// TIA Portal V15.1 export
// export: Created 2024-06-21T08:41:07.4189134Z, ExportSetting WithDefaults, DisplayName Totally Integrated Automation Portal, DisplayVersion V15.1 Update 5, DisplayName TIA Portal Openness, DisplayVersion V15.1 Update 5, DisplayName SINAMICS Startdrive Advanced, DisplayVersion V15.1, DisplayName G130, G150, S120, S150, SINAMICS MV, S210, DisplayVersion V15.1, DisplayName G110M, G120, G120C, G120D, G120P, DisplayVersion V15.1, DisplayName STEP 7 Professional, DisplayVersion V15.1 Update 5, DisplayName STEP 7 Safety, DisplayVersion V15.1, DisplayName WinCC Professional, DisplayVersion V15.1 Update 5, DisplayName SIMATIC Visualization Architect, DisplayVersion V15.1
FUNCTION_BLOCK "LGBKP400"   // FB6660, FBD
TITLE = KP400 handling
{ S7_Optimized_Access := 'FALSE' }
AUTHOR : VCG
FAMILY : OPanel
VERSION : 1.0
// ================================================================================
// This module handles the modezone OP.
// Interlocking between OP's in the same modezone
// User interaction between the modezone and the interface
// ================================================================================
// 2021-07-26
// stored: AutoNumber false, IsIECCheckEnabled false, SetENOAutomatically False, UDAEnableTagReadback false
   VAR_INPUT
      I_OP_ID { ExternalAccessible := 'False'; ExternalVisible := 'False'; ExternalWritable := 'False'} : Int;   // Unique OP identification in the group
      I_ActiveHMI { ExternalAccessible := 'False'; ExternalVisible := 'False'; ExternalWritable := 'False'} : Int;   // Active HMI in the Modeselector
      I_ExtPBSet { ExternalAccessible := 'False'; ExternalVisible := 'False'; ExternalWritable := 'False'} : Bool;   // External PB set
      I_ExtPBReset { ExternalAccessible := 'False'; ExternalVisible := 'False'; ExternalWritable := 'False'} : Bool;   // External PB reset
   END_VAR
   VAR_OUTPUT
      O_ASSelected { ExternalAccessible := 'False'; ExternalVisible := 'False'; ExternalWritable := 'False'} : Bool;
      O_LampTest { ExternalAccessible := 'False'; ExternalVisible := 'False'; ExternalWritable := 'False'} : Bool;
      O_AutoModeSel { ExternalAccessible := 'False'; ExternalVisible := 'False'; ExternalWritable := 'False'} : Bool;
      O_ManualModeSel { ExternalAccessible := 'False'; ExternalVisible := 'False'; ExternalWritable := 'False'} : Bool;
      O_ResetSeq { ExternalAccessible := 'False'; ExternalVisible := 'False'; ExternalWritable := 'False'} : Bool;
      O_Start { ExternalAccessible := 'False'; ExternalVisible := 'False'; ExternalWritable := 'False'} : Bool;
      O_AlarmReset { ExternalAccessible := 'False'; ExternalVisible := 'False'; ExternalWritable := 'False'} : Bool;
      O_HighSpeed { ExternalAccessible := 'False'; ExternalVisible := 'False'; ExternalWritable := 'False'} : Bool;
      O_MovCode { ExternalAccessible := 'False'; ExternalVisible := 'False'; ExternalWritable := 'False'} : Int;
   END_VAR
   VAR_IN_OUT
      IO_GroupInterlock { ExternalAccessible := 'False'; ExternalVisible := 'False'; ExternalWritable := 'False'} : Int;   // Is this OP selected? Refers to the interlocking word of this group
      H_HMI : "H_HMI";
      H_GBKP400 : "H_GBKP400";
      IO_Modes : "Modes";   // Modes IO
   END_VAR
   VAR DB_SPECIFIC
      OP_Selected { ExternalAccessible := 'False'; ExternalVisible := 'False'; ExternalWritable := 'False'} : Bool;
      OP_Selected_NE { ExternalAccessible := 'False'; ExternalVisible := 'False'; ExternalWritable := 'False'} : Bool;
      FK_F1_Pressed { ExternalAccessible := 'False'; ExternalVisible := 'False'; ExternalWritable := 'False'} : Bool;
      FK_F2_Pressed { ExternalAccessible := 'False'; ExternalVisible := 'False'; ExternalWritable := 'False'} : Bool;
      FK_F3_Pressed { ExternalAccessible := 'False'; ExternalVisible := 'False'; ExternalWritable := 'False'} : Bool;
      FK_F4_Pressed { ExternalAccessible := 'False'; ExternalVisible := 'False'; ExternalWritable := 'False'} : Bool;
      FK_F5_Pressed { ExternalAccessible := 'False'; ExternalVisible := 'False'; ExternalWritable := 'False'} : Bool;   // Main Pressed
      FK_F6_Pressed { ExternalAccessible := 'False'; ExternalVisible := 'False'; ExternalWritable := 'False'} : Bool;   // Auto Pressed
      FK_F7_Pressed { ExternalAccessible := 'False'; ExternalVisible := 'False'; ExternalWritable := 'False'} : Bool;   // Man Pressed
      FK_F8_Pressed { ExternalAccessible := 'False'; ExternalVisible := 'False'; ExternalWritable := 'False'} : Bool;   // Step Pressed
      FK_F1_Pressed_hPE { ExternalAccessible := 'False'; ExternalVisible := 'False'; ExternalWritable := 'False'} : Bool;
      FK_F2_Pressed_hPE { ExternalAccessible := 'False'; ExternalVisible := 'False'; ExternalWritable := 'False'} : Bool;
      FK_F3_Pressed_hPE { ExternalAccessible := 'False'; ExternalVisible := 'False'; ExternalWritable := 'False'} : Bool;
      FK_F4_Pressed_hPE { ExternalAccessible := 'False'; ExternalVisible := 'False'; ExternalWritable := 'False'} : Bool;
      FK_F5_Pressed_hPE { ExternalAccessible := 'False'; ExternalVisible := 'False'; ExternalWritable := 'False'} : Bool;
      FK_F6_Pressed_hPE { ExternalAccessible := 'False'; ExternalVisible := 'False'; ExternalWritable := 'False'} : Bool;
      FK_F7_Pressed_hPE { ExternalAccessible := 'False'; ExternalVisible := 'False'; ExternalWritable := 'False'} : Bool;
      FK_F8_Pressed_hPE { ExternalAccessible := 'False'; ExternalVisible := 'False'; ExternalWritable := 'False'} : Bool;
      FK_F1_Pressed_PE { ExternalAccessible := 'False'; ExternalVisible := 'False'; ExternalWritable := 'False'} : Bool;
      FK_F2_Pressed_PE { ExternalAccessible := 'False'; ExternalVisible := 'False'; ExternalWritable := 'False'} : Bool;
      FK_F3_Pressed_PE { ExternalAccessible := 'False'; ExternalVisible := 'False'; ExternalWritable := 'False'} : Bool;
      FK_F4_Pressed_PE { ExternalAccessible := 'False'; ExternalVisible := 'False'; ExternalWritable := 'False'} : Bool;
      FK_F5_Pressed_PE { ExternalAccessible := 'False'; ExternalVisible := 'False'; ExternalWritable := 'False'} : Bool;
      FK_F6_Pressed_PE { ExternalAccessible := 'False'; ExternalVisible := 'False'; ExternalWritable := 'False'} : Bool;
      FK_F7_Pressed_PE { ExternalAccessible := 'False'; ExternalVisible := 'False'; ExternalWritable := 'False'} : Bool;
      FK_F8_Pressed_PE { ExternalAccessible := 'False'; ExternalVisible := 'False'; ExternalWritable := 'False'} : Bool;
      MainScreenActive { ExternalAccessible := 'False'; ExternalVisible := 'False'; ExternalWritable := 'False'} : Bool;
      AutoScreenActive { ExternalAccessible := 'False'; ExternalVisible := 'False'; ExternalWritable := 'False'} : Bool;
      AutoSelScreenActive { ExternalAccessible := 'False'; ExternalVisible := 'False'; ExternalWritable := 'False'} : Bool;
      ManScreenActive { ExternalAccessible := 'False'; ExternalVisible := 'False'; ExternalWritable := 'False'} : Bool;
      MVTScreenActive { ExternalAccessible := 'False'; ExternalVisible := 'False'; ExternalWritable := 'False'} : Bool;
      ProdScreenActive { ExternalAccessible := 'False'; ExternalVisible := 'False'; ExternalWritable := 'False'} : Bool;
      SSScreenActive { ExternalAccessible := 'False'; ExternalVisible := 'False'; ExternalWritable := 'False'} : Bool;
      SSSelScreenActive { ExternalAccessible := 'False'; ExternalVisible := 'False'; ExternalWritable := 'False'} : Bool;
      Request_Logout { ExternalAccessible := 'False'; ExternalVisible := 'False'; ExternalWritable := 'False'} : Bool;
      OP_TimeoutInput { ExternalAccessible := 'False'; ExternalVisible := 'False'; ExternalWritable := 'False'} : Bool;
      AutoSel { ExternalAccessible := 'False'; ExternalVisible := 'False'; ExternalWritable := 'False'} : Bool;
      ManualSel { ExternalAccessible := 'False'; ExternalVisible := 'False'; ExternalWritable := 'False'} : Bool;
      AutoSel_PE { ExternalAccessible := 'False'; ExternalVisible := 'False'; ExternalWritable := 'False'} : Bool;
      ManSel_PE { ExternalAccessible := 'False'; ExternalVisible := 'False'; ExternalWritable := 'False'} : Bool;
      AlarmReset { ExternalAccessible := 'False'; ExternalVisible := 'False'; ExternalWritable := 'False'} : Bool;
      Start { ExternalAccessible := 'False'; ExternalVisible := 'False'; ExternalWritable := 'False'} : Bool;
      ResetTM { ExternalAccessible := 'False'; ExternalVisible := 'False'; ExternalWritable := 'False'} : Bool;
      ResetSeq { ExternalAccessible := 'False'; ExternalVisible := 'False'; ExternalWritable := 'False'} : Bool;
      AutoMode { ExternalAccessible := 'False'; ExternalVisible := 'False'; ExternalWritable := 'False'} : Bool;
      StepMode { ExternalAccessible := 'False'; ExternalVisible := 'False'; ExternalWritable := 'False'} : Bool;
      ManualMode { ExternalAccessible := 'False'; ExternalVisible := 'False'; ExternalWritable := 'False'} : Bool;
      Alarm { ExternalAccessible := 'False'; ExternalVisible := 'False'; ExternalWritable := 'False'} : Bool;
      STAT4 { ExternalAccessible := 'False'; ExternalVisible := 'False'; ExternalWritable := 'False'} : Bool;
      STAT5 { ExternalAccessible := 'False'; ExternalVisible := 'False'; ExternalWritable := 'False'} : Bool;
      STAT6 { ExternalAccessible := 'False'; ExternalVisible := 'False'; ExternalWritable := 'False'} : Bool;
      STAT7 { ExternalAccessible := 'False'; ExternalVisible := 'False'; ExternalWritable := 'False'} : Bool;
      STAT8 { ExternalAccessible := 'False'; ExternalVisible := 'False'; ExternalWritable := 'False'} : Bool;
      STAT9 { ExternalAccessible := 'False'; ExternalVisible := 'False'; ExternalWritable := 'False'} : Bool;
      STAT10 { ExternalAccessible := 'False'; ExternalVisible := 'False'; ExternalWritable := 'False'} : Bool;
      STAT11 { ExternalAccessible := 'False'; ExternalVisible := 'False'; ExternalWritable := 'False'} : Bool;
      STAT12 { ExternalAccessible := 'False'; ExternalVisible := 'False'; ExternalWritable := 'False'} : Bool;
      OP_ScreenWanted { ExternalAccessible := 'False'; ExternalVisible := 'False'; ExternalWritable := 'False'} : Int;
      MovCode { ExternalAccessible := 'False'; ExternalVisible := 'False'; ExternalWritable := 'False'} : Int;
      MovCodeCalculation { ExternalAccessible := 'False'; ExternalVisible := 'False'; ExternalWritable := 'False'} : Int;
      ProdStatus { ExternalAccessible := 'False'; ExternalVisible := 'False'; ExternalWritable := 'False'} : Int;   // Production Mode
      ActiveMode { ExternalAccessible := 'False'; ExternalVisible := 'False'; ExternalWritable := 'False'} : Int;
      OPMode { ExternalAccessible := 'False'; ExternalVisible := 'False'; ExternalWritable := 'False'} : Int;
      GroupInterlock { ExternalAccessible := 'False'; ExternalVisible := 'False'; ExternalWritable := 'False'} : Int;
      ResetOP { ExternalAccessible := 'False'; ExternalVisible := 'False'; ExternalWritable := 'False'} : Bool;
      Edge { ExternalAccessible := 'False'; ExternalVisible := 'False'; ExternalWritable := 'False'} : Array[1..10] of Bool;
   END_VAR
   VAR
      Timer_Timeout_Input { ExternalAccessible := 'False'; ExternalVisible := 'False'; ExternalWritable := 'False'} : "LTimer";
   END_VAR
   VAR DB_SPECIFIC
      ModeEdge { ExternalAccessible := 'False'; ExternalVisible := 'False'; ExternalWritable := 'False'} : Array[1..10] of Bool;
   END_VAR
   VAR_TEMP
      OP_CommsDB : Int;
   END_VAR
   // // H_GBKP400.OPStatus : KP400 status
   // // H_GBKP400.OPMode : KP400 mode
   // // H_GBKP400.OPAdditional : KP400 additional info
   VAR_TEMP   // added for the SCL form of the ladder/FBD networks
      _w1 : Bool;
   END_VAR
BEGIN

REGION Network 1: **** 1 - Inputs **** Is this KP400 active?
   // Is this KP400 active?
   // IF yes:
   //  * Set OP as active 
   // IF not:
   //  * Reset flowcode
   //  * Reset MVT code
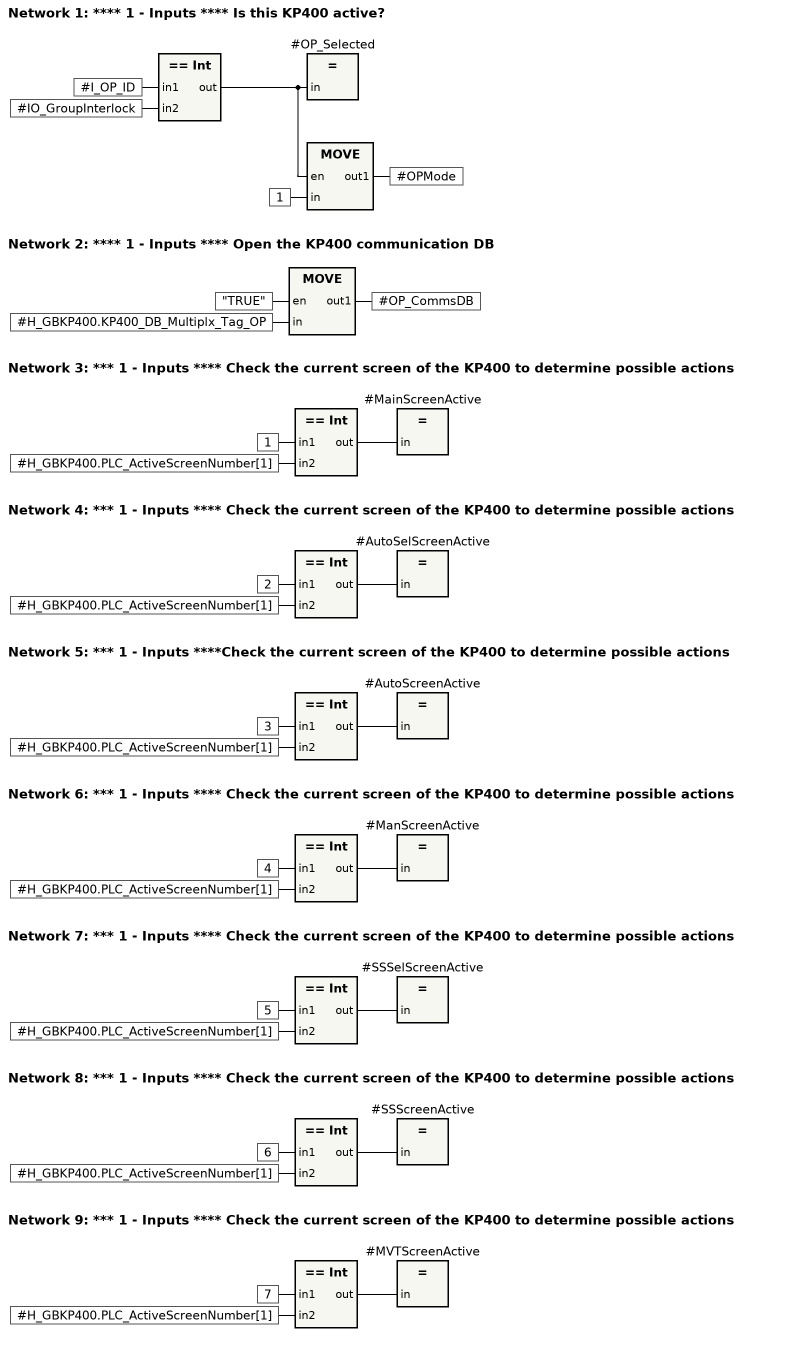
   #OP_Selected := #I_OP_ID = #IO_GroupInterlock;
   IF #OP_Selected THEN #OPMode := 1; END_IF;
END_REGION

REGION Network 2: **** 1 - Inputs **** Open the KP400 communication DB
   // Open the KP400 communication DB
   IF "TRUE" THEN #OP_CommsDB := #H_GBKP400.KP400_DB_Multiplx_Tag_OP; END_IF;
END_REGION

REGION Network 3: *** 1 - Inputs **** Check the current screen of the KP400 to determine possible actions
   // Check the current screen of the KP400 to determine possible actions
   //  1: Menu_Main
   //  2: Menu_Auto_Sel
   //  3: Menu_Auto
   //  4: Menu_Man
   //  5: Menu_SS_Sel
   //  6: Menu_SS
   //  7: Menu_MVT
   //  8: Menu_Flow
   //  9: Menu_Prod
   #MainScreenActive := 1 = #H_GBKP400.PLC_ActiveScreenNumber[1];
END_REGION

REGION Network 4: *** 1 - Inputs **** Check the current screen of the KP400 to determine possible actions
   // Check the current screen of the KP400 to determine possible actions
   //  2: Menu_Auto_Sel
   #AutoSelScreenActive := 2 = #H_GBKP400.PLC_ActiveScreenNumber[1];
END_REGION

REGION Network 5: *** 1 - Inputs ****Check the current screen of the KP400 to determine possible actions
   // Check the current screen of the KP400  to determine possible actions
   //  3: Menu_Auto
   #AutoScreenActive := 3 = #H_GBKP400.PLC_ActiveScreenNumber[1];
END_REGION

REGION Network 6: *** 1 - Inputs **** Check the current screen of the KP400 to determine possible actions
   // Check the current screen of the KP400  to determine possible actions
   //  4: Menu_Man
   #ManScreenActive := 4 = #H_GBKP400.PLC_ActiveScreenNumber[1];
END_REGION

REGION Network 7: *** 1 - Inputs **** Check the current screen of the KP400 to determine possible actions
   // Check the current screen of the KP400  to determine possible actions
   //  5: Menu_SS_Sel
   #SSSelScreenActive := 5 = #H_GBKP400.PLC_ActiveScreenNumber[1];
END_REGION

REGION Network 8: *** 1 - Inputs **** Check the current screen of the KP400 to determine possible actions
   // Check the current screen of the KP400  to determine possible actions
   //  6: Menu_SS
   #SSScreenActive := 6 = #H_GBKP400.PLC_ActiveScreenNumber[1];
END_REGION

REGION Network 9: *** 1 - Inputs **** Check the current screen of the KP400 to determine possible actions
   // Check the current screen of the KP400  to determine possible actions
   //  7: Menu_MVT
   #MVTScreenActive := 7 = #H_GBKP400.PLC_ActiveScreenNumber[1];
END_REGION

REGION Network 10: *** 1 - Inputs **** Check the current screen of the KP400 to determine possible actions
   // Check the current screen of the KP400  to determine possible actions
   //  9: Menu_Prod
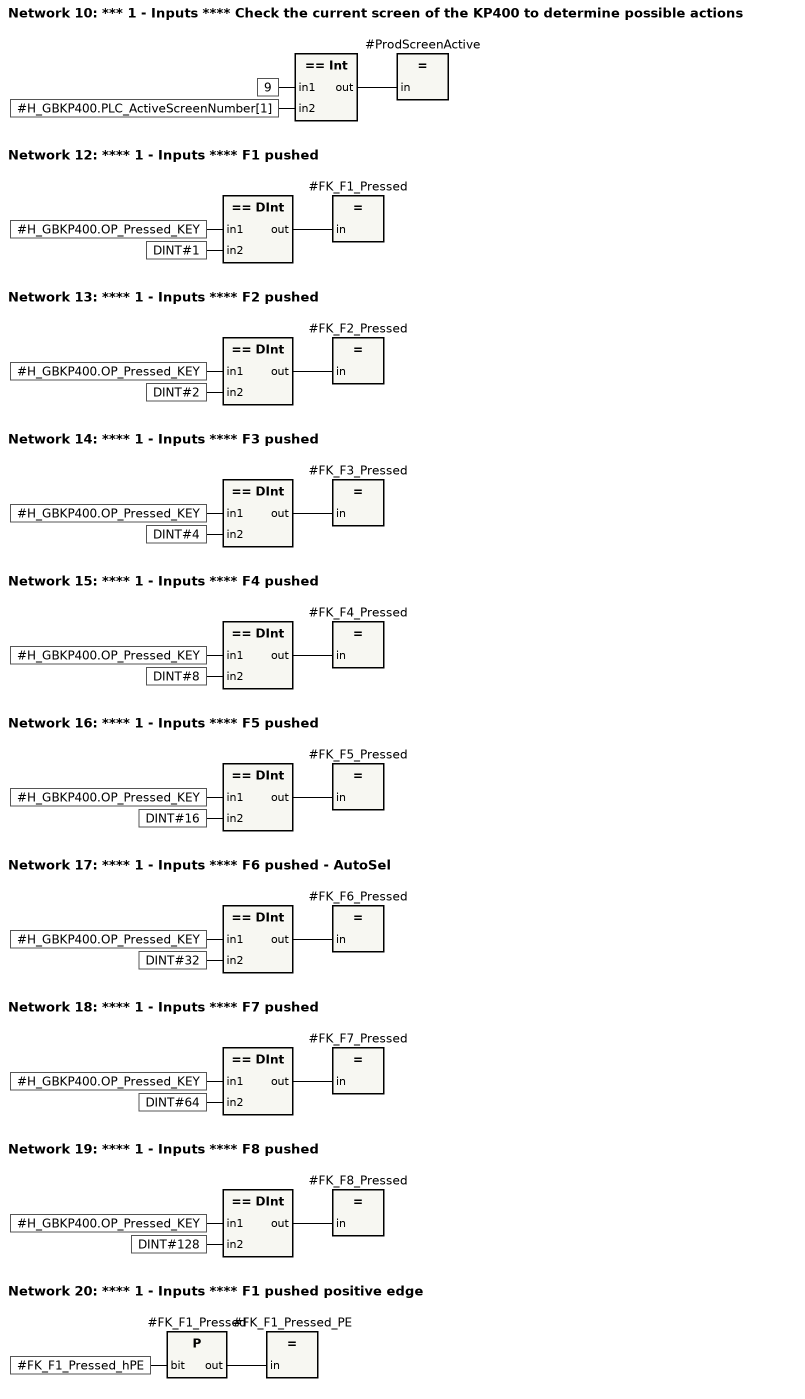
   #ProdScreenActive := 9 = #H_GBKP400.PLC_ActiveScreenNumber[1];
END_REGION

NETWORK
TITLE = **** 1 - Inputs **** Handling of the push buttons F1-F4
// Handling of the push buttons F1-F4 on the OP; these are the only ones that 
// interact with the PLC, for every key the 'press' detection and the edge 
// detection
      NOP   0;


REGION Network 12: **** 1 - Inputs **** F1 pushed
   // F1 pushed
   #FK_F1_Pressed := #H_GBKP400.OP_Pressed_KEY = DINT#1;
END_REGION

REGION Network 13: **** 1 - Inputs **** F2 pushed
   // F2 pushed
   #FK_F2_Pressed := #H_GBKP400.OP_Pressed_KEY = DINT#2;
END_REGION

REGION Network 14: **** 1 - Inputs **** F3 pushed
   // F3 pushed
   #FK_F3_Pressed := #H_GBKP400.OP_Pressed_KEY = DINT#4;
END_REGION

REGION Network 15: **** 1 - Inputs **** F4 pushed
   // F4 pushed
   #FK_F4_Pressed := #H_GBKP400.OP_Pressed_KEY = DINT#8;
END_REGION

REGION Network 16: **** 1 - Inputs **** F5 pushed
   // F5 pushed
   #FK_F5_Pressed := #H_GBKP400.OP_Pressed_KEY = DINT#16;
END_REGION

REGION Network 17: **** 1 - Inputs **** F6 pushed - AutoSel
   // F6 pushed
   #FK_F6_Pressed := #H_GBKP400.OP_Pressed_KEY = DINT#32;
END_REGION

REGION Network 18: **** 1 - Inputs **** F7 pushed
   // F7 pushed
   #FK_F7_Pressed := #H_GBKP400.OP_Pressed_KEY = DINT#64;
END_REGION

REGION Network 19: **** 1 - Inputs **** F8 pushed
   // F8 pushed
   #FK_F8_Pressed := #H_GBKP400.OP_Pressed_KEY = DINT#128;
END_REGION

REGION Network 20: **** 1 - Inputs **** F1 pushed positive edge
   // F1 pushed positive edge detection
   #_w1 := #FK_F1_Pressed AND NOT #FK_F1_Pressed_hPE;   // rising edge of #FK_F1_Pressed
   #FK_F1_Pressed_hPE := #FK_F1_Pressed;
   #FK_F1_Pressed_PE := #_w1;
END_REGION

REGION Network 21: **** 1 - Inputs **** F2 pushed positive edge
   // F2 pushed positive edge detection
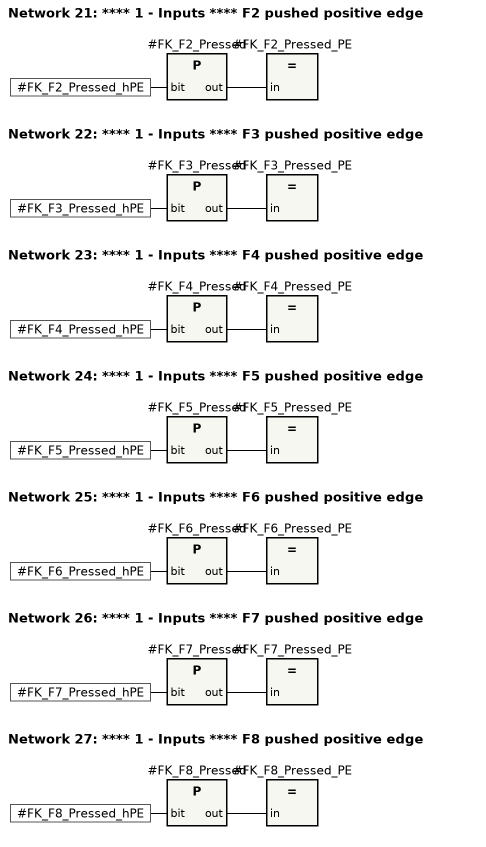
   #_w1 := #FK_F2_Pressed AND NOT #FK_F2_Pressed_hPE;   // rising edge of #FK_F2_Pressed
   #FK_F2_Pressed_hPE := #FK_F2_Pressed;
   #FK_F2_Pressed_PE := #_w1;
END_REGION

REGION Network 22: **** 1 - Inputs **** F3 pushed positive edge
   // F3 pushed positive edge detection
   #_w1 := #FK_F3_Pressed AND NOT #FK_F3_Pressed_hPE;   // rising edge of #FK_F3_Pressed
   #FK_F3_Pressed_hPE := #FK_F3_Pressed;
   #FK_F3_Pressed_PE := #_w1;
END_REGION

REGION Network 23: **** 1 - Inputs **** F4 pushed positive edge
   // F4 pushed positive edge detection
   #_w1 := #FK_F4_Pressed AND NOT #FK_F4_Pressed_hPE;   // rising edge of #FK_F4_Pressed
   #FK_F4_Pressed_hPE := #FK_F4_Pressed;
   #FK_F4_Pressed_PE := #_w1;
END_REGION

REGION Network 24: **** 1 - Inputs **** F5 pushed positive edge
   // F5 pushed positive edge detection
   #_w1 := #FK_F5_Pressed AND NOT #FK_F5_Pressed_hPE;   // rising edge of #FK_F5_Pressed
   #FK_F5_Pressed_hPE := #FK_F5_Pressed;
   #FK_F5_Pressed_PE := #_w1;
END_REGION

REGION Network 25: **** 1 - Inputs **** F6 pushed positive edge
   // F6 pushed positive edge detection
   #_w1 := #FK_F6_Pressed AND NOT #FK_F6_Pressed_hPE;   // rising edge of #FK_F6_Pressed
   #FK_F6_Pressed_hPE := #FK_F6_Pressed;
   #FK_F6_Pressed_PE := #_w1;
END_REGION

REGION Network 26: **** 1 - Inputs **** F7 pushed positive edge
   // F7 pushed positive edge detection
   #_w1 := #FK_F7_Pressed AND NOT #FK_F7_Pressed_hPE;   // rising edge of #FK_F7_Pressed
   #FK_F7_Pressed_hPE := #FK_F7_Pressed;
   #FK_F7_Pressed_PE := #_w1;
END_REGION

REGION Network 27: **** 1 - Inputs **** F8 pushed positive edge
   // F8 pushed positive edge detection
   #_w1 := #FK_F8_Pressed AND NOT #FK_F8_Pressed_hPE;   // rising edge of #FK_F8_Pressed
   #FK_F8_Pressed_hPE := #FK_F8_Pressed;
   #FK_F8_Pressed_PE := #_w1;
END_REGION

REGION Network 28: **** 1 - Inputs **** Evaluate current mode
   // Evaluate current mode
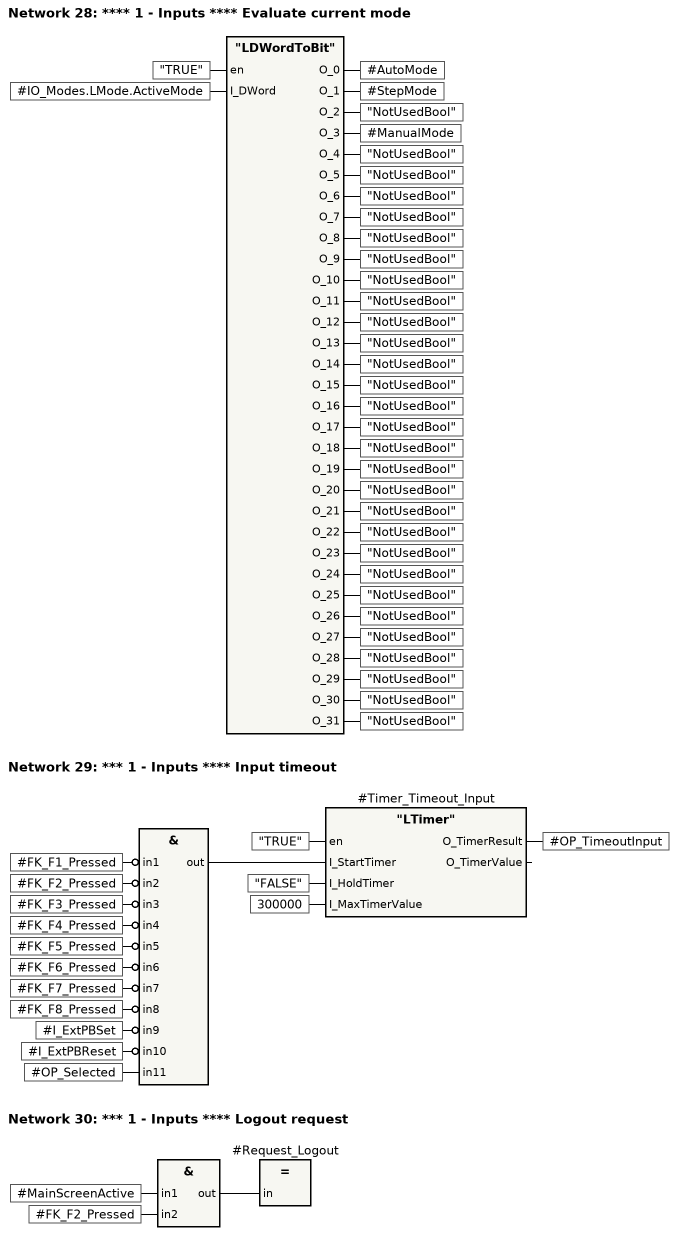
   IF "TRUE" THEN
       "LDWordToBit"(I_DWord := #IO_Modes.LMode.ActiveMode,
                     O_0 => #AutoMode,
                     O_1 => #StepMode,
                     O_2 => "NotUsedBool",
                     O_3 => #ManualMode,
                     O_4 => "NotUsedBool",
                     O_5 => "NotUsedBool",
                     O_6 => "NotUsedBool",
                     O_7 => "NotUsedBool",
                     O_8 => "NotUsedBool",
                     O_9 => "NotUsedBool",
                     O_10 => "NotUsedBool",
                     O_11 => "NotUsedBool",
                     O_12 => "NotUsedBool",
                     O_13 => "NotUsedBool",
                     O_14 => "NotUsedBool",
                     O_15 => "NotUsedBool",
                     O_16 => "NotUsedBool",
                     O_17 => "NotUsedBool",
                     O_18 => "NotUsedBool",
                     O_19 => "NotUsedBool",
                     O_20 => "NotUsedBool",
                     O_21 => "NotUsedBool",
                     O_22 => "NotUsedBool",
                     O_23 => "NotUsedBool",
                     O_24 => "NotUsedBool",
                     O_25 => "NotUsedBool",
                     O_26 => "NotUsedBool",
                     O_27 => "NotUsedBool",
                     O_28 => "NotUsedBool",
                     O_29 => "NotUsedBool",
                     O_30 => "NotUsedBool",
                     O_31 => "NotUsedBool");
   END_IF;
END_REGION

REGION Network 29: *** 1 - Inputs **** Input timeout
   // Input timeout
   IF "TRUE" THEN
       #Timer_Timeout_Input(I_StartTimer := NOT #FK_F1_Pressed AND NOT #FK_F2_Pressed AND NOT #FK_F3_Pressed AND NOT #FK_F4_Pressed AND NOT #FK_F5_Pressed AND NOT #FK_F6_Pressed AND NOT #FK_F7_Pressed AND NOT #FK_F8_Pressed AND NOT #I_ExtPBSet AND NOT #I_ExtPBReset AND #OP_Selected,   // "LTimer"
                            I_HoldTimer := "FALSE",
                            I_MaxTimerValue := 300000,
                            O_TimerResult => #OP_TimeoutInput);
   END_IF;
END_REGION

REGION Network 30: *** 1 - Inputs **** Logout request
   // Logout request
   // Main menu and F2
   #Request_Logout := #MainScreenActive AND #FK_F2_Pressed;
END_REGION

REGION Network 31: *** 4.4 Machine Status, calculated *** Set movement code
   // Set movement code
   // Reset movement code to 999 if the MVT menu is left
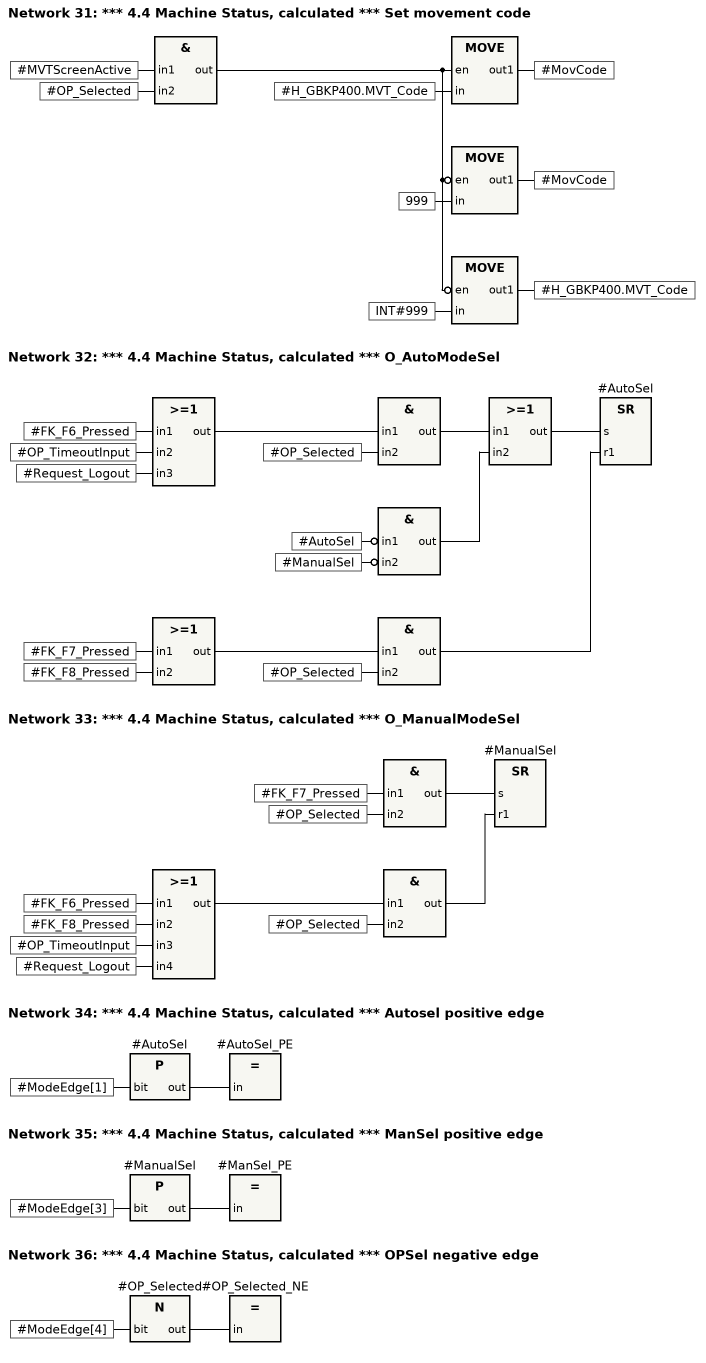
   #_w1 := #MVTScreenActive AND #OP_Selected;
   IF #_w1 THEN #MovCode := #H_GBKP400.MVT_Code; END_IF;
   IF NOT #_w1 THEN
       #MovCode := 999;
       #H_GBKP400.MVT_Code := INT#999;
   END_IF;
END_REGION

REGION Network 32: *** 4.4 Machine Status, calculated *** O_AutoModeSel
   // O_AutoModeSel
   IF ((#FK_F6_Pressed OR #OP_TimeoutInput OR #Request_Logout) AND #OP_Selected) OR (NOT #AutoSel AND NOT #ManualSel) THEN
       #AutoSel := TRUE;   // SR flip-flop
   END_IF;
   IF (#FK_F7_Pressed OR #FK_F8_Pressed) AND #OP_Selected THEN #AutoSel := FALSE; END_IF;
END_REGION

REGION Network 33: *** 4.4 Machine Status, calculated *** O_ManualModeSel
   // O_ManualModeSel
   IF #FK_F7_Pressed AND #OP_Selected THEN
       #ManualSel := TRUE;   // SR flip-flop
   END_IF;
   IF (#FK_F6_Pressed OR #FK_F8_Pressed OR #OP_TimeoutInput OR #Request_Logout) AND #OP_Selected THEN
       #ManualSel := FALSE;
   END_IF;
END_REGION

REGION Network 34: *** 4.4 Machine Status, calculated *** Autosel positive edge
   #_w1 := #AutoSel AND NOT #ModeEdge[1];   // rising edge of #AutoSel
   #ModeEdge[1] := #AutoSel;
   #AutoSel_PE := #_w1;
END_REGION

REGION Network 35: *** 4.4 Machine Status, calculated *** ManSel positive edge
   #_w1 := #ManualSel AND NOT #ModeEdge[3];   // rising edge of #ManualSel
   #ModeEdge[3] := #ManualSel;
   #ManSel_PE := #_w1;
END_REGION

REGION Network 36: *** 4.4 Machine Status, calculated *** OPSel negative edge
   #_w1 := NOT #OP_Selected AND #ModeEdge[4];   // falling edge of #OP_Selected
   #ModeEdge[4] := #OP_Selected;
   #OP_Selected_NE := #_w1;
END_REGION

REGION Network 37: *** 4.4 Machine Status, calculated *** O_ResetSeq
   // O_ResetSeq
   //  * K3 AND
   //  * Menu_Man            OR
   //  * Menu_MVT_Selected   
   // 
   // O_ResetTM identical to O_ResetSeq
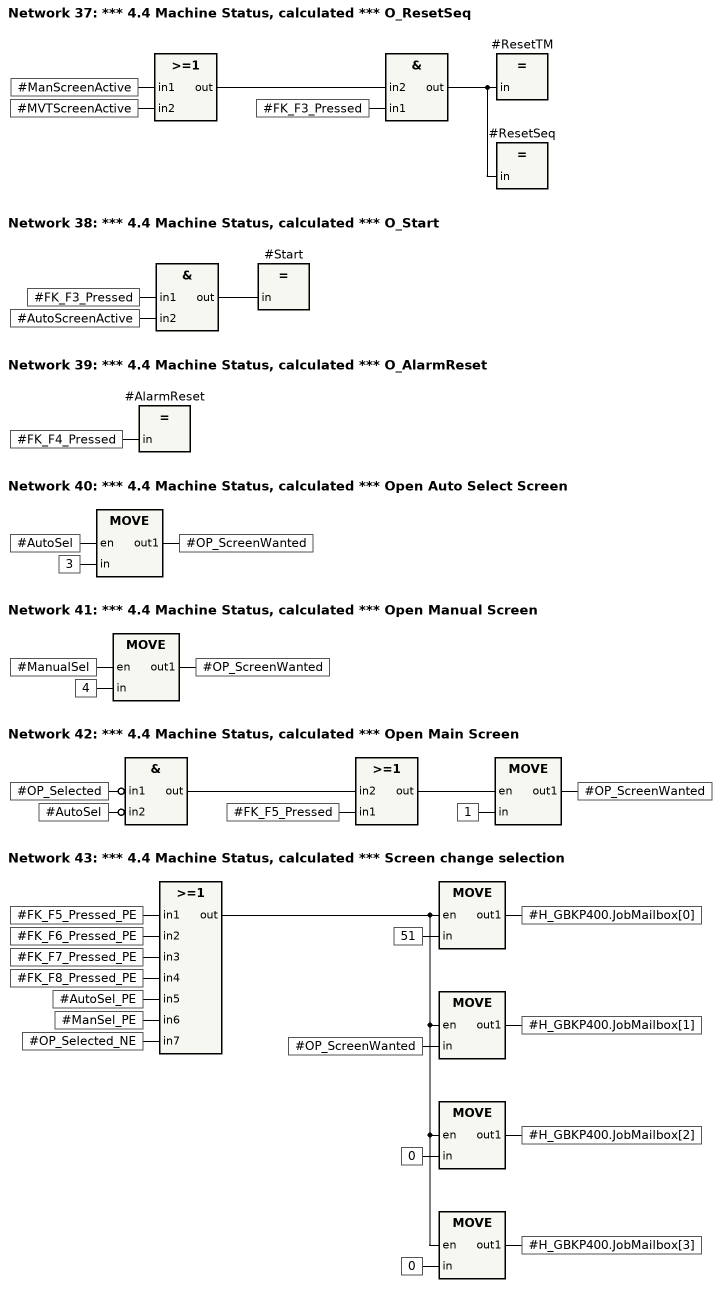
   #ResetTM := (#ManScreenActive OR #MVTScreenActive) AND #FK_F3_Pressed;
   #ResetSeq := #ResetTM;
END_REGION

REGION Network 38: *** 4.4 Machine Status, calculated *** O_Start
   // O_Start
   //  * K3 AND
   //  * Menu_Auto_Selected  OR
   //  * Menu_SS_Selected
   #Start := #FK_F3_Pressed AND #AutoScreenActive;
END_REGION

REGION Network 39: *** 4.4 Machine Status, calculated *** O_AlarmReset
   // O_AlarmReset
   //  * K4 AND
   //  * Menu_Main           OR
   //  * Menu_Auto           OR
   //  * Menu_Auto_Selected  OR
   //  * Menu_SS             OR
   //  * Menu_SS_Selected    OR
   //  * Menu_Man            OR
   //  * Menu_MVT_Selected
   #AlarmReset := #FK_F4_Pressed;
END_REGION

REGION Network 40: *** 4.4 Machine Status, calculated *** Open Auto Select Screen
   // Open Auto Select Screen
   IF #AutoSel THEN #OP_ScreenWanted := 3; END_IF;
END_REGION

REGION Network 41: *** 4.4 Machine Status, calculated *** Open Manual Screen
   // Open Manual Screen
   IF #ManualSel THEN #OP_ScreenWanted := 4; END_IF;
END_REGION

REGION Network 42: *** 4.4 Machine Status, calculated *** Open Main Screen
   // Open Main Screen
   IF (NOT #OP_Selected AND NOT #AutoSel) OR #FK_F5_Pressed THEN #OP_ScreenWanted := 1; END_IF;
END_REGION

REGION Network 43: *** 4.4 Machine Status, calculated *** Screen change selection
   // Open StepStep Screen
   IF #FK_F5_Pressed_PE OR #FK_F6_Pressed_PE OR #FK_F7_Pressed_PE OR #FK_F8_Pressed_PE OR #AutoSel_PE OR #ManSel_PE OR #OP_Selected_NE THEN
       #H_GBKP400.JobMailbox[0] := 51;
       #H_GBKP400.JobMailbox[1] := #OP_ScreenWanted;
       #H_GBKP400.JobMailbox[2] := 0;
       #H_GBKP400.JobMailbox[3] := 0;
   END_IF;
END_REGION

REGION Network 44: *** 4.4 Machine Status, calculated *** Set the op status to locked
   // Set the op status to locked
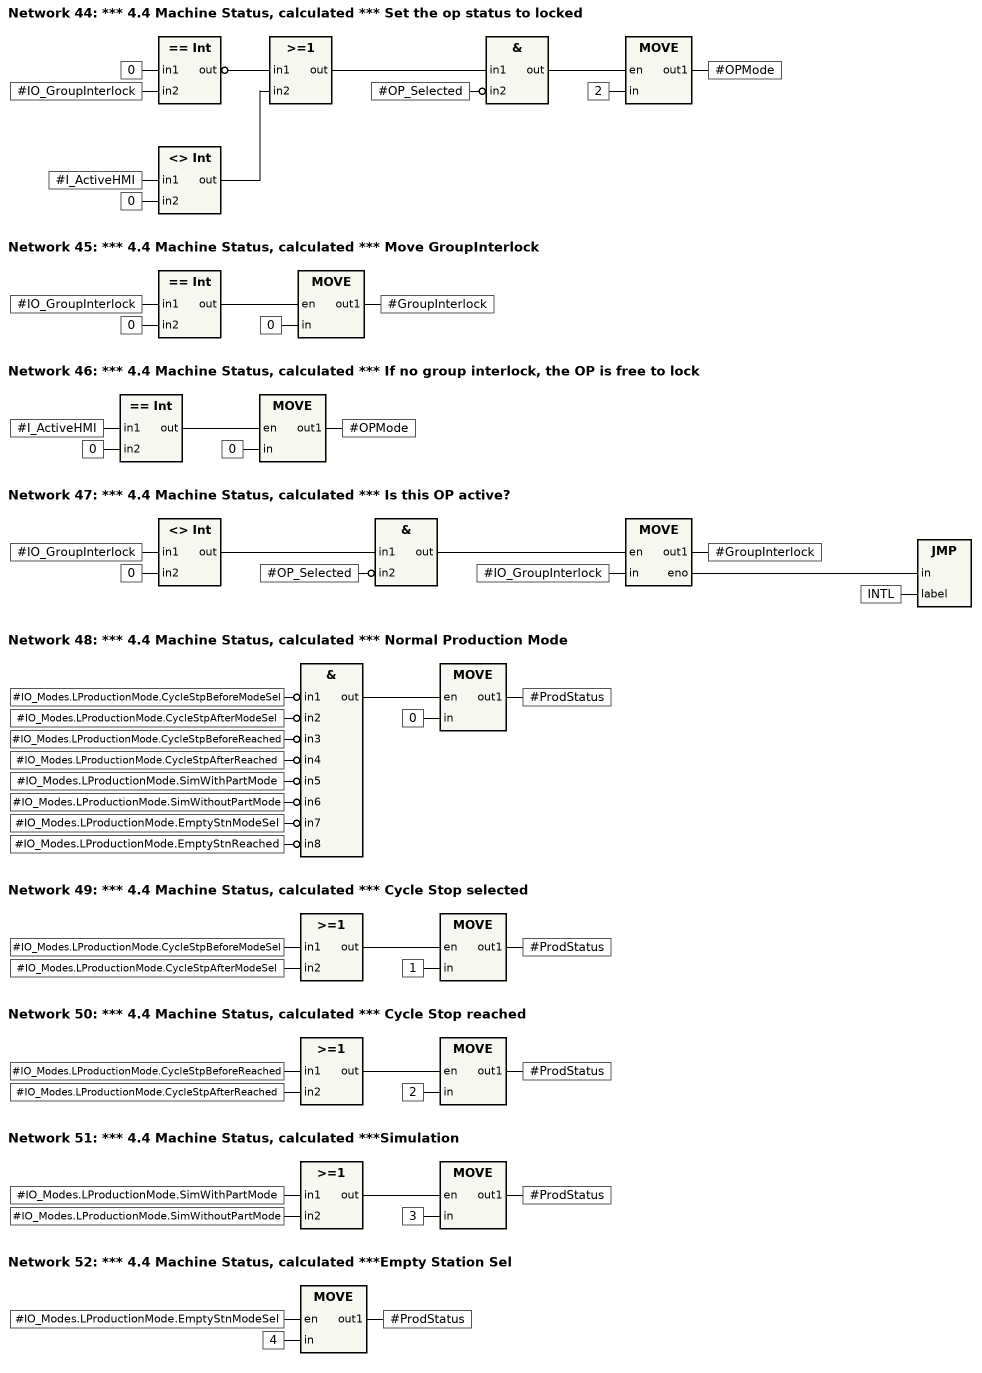
   IF (NOT (0 = #IO_GroupInterlock) OR (#I_ActiveHMI <> 0)) AND NOT #OP_Selected THEN #OPMode := 2; END_IF;
END_REGION

REGION Network 45: *** 4.4 Machine Status, calculated *** Move GroupInterlock
   // If no group interlock, the OP is free to lock
   IF #IO_GroupInterlock = 0 THEN #GroupInterlock := 0; END_IF;
END_REGION

REGION Network 46: *** 4.4 Machine Status, calculated *** If no group interlock, the OP is free to lock
   // If no group interlock, the OP is free to lock
   IF #I_ActiveHMI = 0 THEN #OPMode := 0; END_IF;
END_REGION

REGION Network 47: *** 4.4 Machine Status, calculated *** Is this OP active?
   // Is this OP active?
   // ENO of a box is taken as its EN; it also drops when the box reports an error
   #_w1 := (#IO_GroupInterlock <> 0) AND NOT #OP_Selected;
   IF #_w1 THEN
       #GroupInterlock := #IO_GroupInterlock;
       GOTO INTL;
   END_IF;
END_REGION

REGION Network 48: *** 4.4 Machine Status, calculated *** Normal Production Mode
   // Normal Production Mode
   IF NOT #IO_Modes.LProductionMode.CycleStpBeforeModeSel AND NOT #IO_Modes.LProductionMode.CycleStpAfterModeSel AND NOT #IO_Modes.LProductionMode.CycleStpBeforeReached AND NOT #IO_Modes.LProductionMode.CycleStpAfterReached AND NOT #IO_Modes.LProductionMode.SimWithPartMode AND NOT #IO_Modes.LProductionMode.SimWithoutPartMode AND NOT #IO_Modes.LProductionMode.EmptyStnModeSel AND NOT #IO_Modes.LProductionMode.EmptyStnReached THEN
       #ProdStatus := 0;
   END_IF;
END_REGION

REGION Network 49: *** 4.4 Machine Status, calculated *** Cycle Stop selected
   // Cycle Stop selected
   IF #IO_Modes.LProductionMode.CycleStpBeforeModeSel OR #IO_Modes.LProductionMode.CycleStpAfterModeSel THEN
       #ProdStatus := 1;
   END_IF;
END_REGION

REGION Network 50: *** 4.4 Machine Status, calculated *** Cycle Stop reached
   // Cycle Stop reached
   IF #IO_Modes.LProductionMode.CycleStpBeforeReached OR #IO_Modes.LProductionMode.CycleStpAfterReached THEN
       #ProdStatus := 2;
   END_IF;
END_REGION

REGION Network 51: *** 4.4 Machine Status, calculated ***Simulation
   // Simulation
   IF #IO_Modes.LProductionMode.SimWithPartMode OR #IO_Modes.LProductionMode.SimWithoutPartMode THEN
       #ProdStatus := 3;
   END_IF;
END_REGION

REGION Network 52: *** 4.4 Machine Status, calculated ***Empty Station Sel
   // Empty Station Sel
   IF #IO_Modes.LProductionMode.EmptyStnModeSel THEN #ProdStatus := 4; END_IF;
END_REGION

REGION Network 53: *** 4.4 Machine Status, calculated ***Empty Station Reached
   // Empty Station Reached
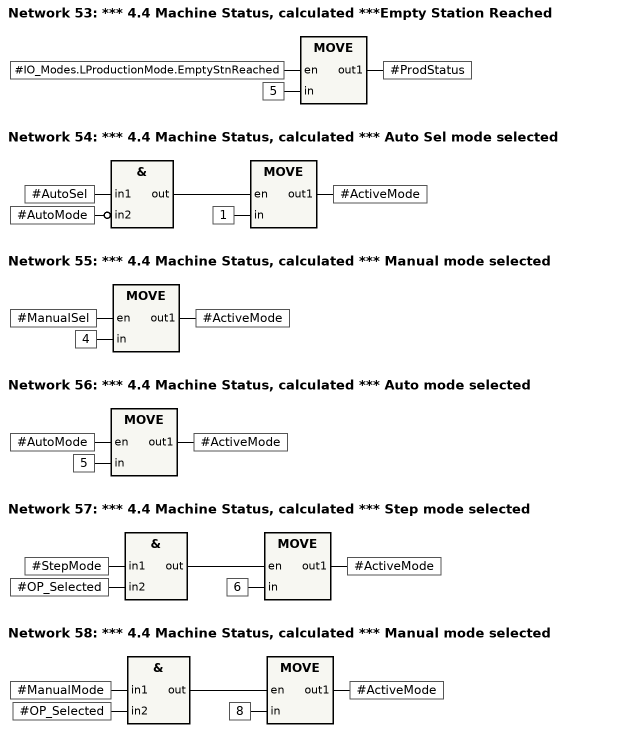
   IF #IO_Modes.LProductionMode.EmptyStnReached THEN #ProdStatus := 5; END_IF;
END_REGION

REGION Network 54: *** 4.4 Machine Status, calculated *** Auto Sel mode selected
   // Auto sel mode selected
   IF #AutoSel AND NOT #AutoMode THEN #ActiveMode := 1; END_IF;
END_REGION

REGION Network 55: *** 4.4 Machine Status, calculated *** Manual mode selected
   // Manual mode selected
   IF #ManualSel THEN #ActiveMode := 4; END_IF;
END_REGION

REGION Network 56: *** 4.4 Machine Status, calculated *** Auto mode selected
   // Auto mode selected
   IF #AutoMode THEN #ActiveMode := 5; END_IF;
END_REGION

REGION Network 57: *** 4.4 Machine Status, calculated *** Step mode selected
   // Step mode selected
   IF #StepMode AND #OP_Selected THEN #ActiveMode := 6; END_IF;
END_REGION

REGION Network 58: *** 4.4 Machine Status, calculated *** Manual mode selected
   // Manual mode selected
   IF #ManualMode AND #OP_Selected THEN #ActiveMode := 8; END_IF;
END_REGION

REGION Network 59: **** 4.6 - Machine status - Indications **** Icon animation
   // Icon animation
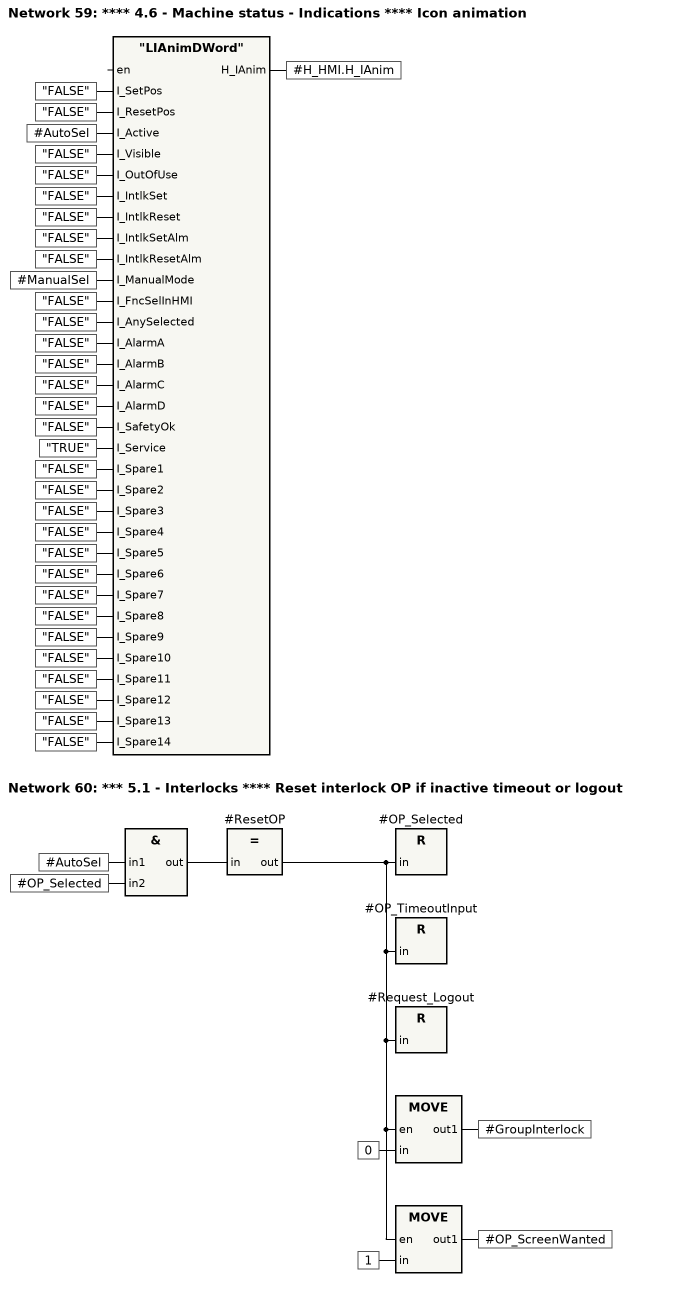
   "LIAnimDWord"(I_SetPos := "FALSE",
                 I_ResetPos := "FALSE",
                 I_Active := #AutoSel,
                 I_Visible := "FALSE",
                 I_OutOfUse := "FALSE",
                 I_IntlkSet := "FALSE",
                 I_IntlkReset := "FALSE",
                 I_IntlkSetAlm := "FALSE",
                 I_IntlkResetAlm := "FALSE",
                 I_ManualMode := #ManualSel,
                 I_FncSelInHMI := "FALSE",
                 I_AnySelected := "FALSE",
                 I_AlarmA := "FALSE",
                 I_AlarmB := "FALSE",
                 I_AlarmC := "FALSE",
                 I_AlarmD := "FALSE",
                 I_SafetyOk := "FALSE",
                 I_Service := "TRUE",
                 I_Spare1 := "FALSE",
                 I_Spare2 := "FALSE",
                 I_Spare3 := "FALSE",
                 I_Spare4 := "FALSE",
                 I_Spare5 := "FALSE",
                 I_Spare6 := "FALSE",
                 I_Spare7 := "FALSE",
                 I_Spare8 := "FALSE",
                 I_Spare9 := "FALSE",
                 I_Spare10 := "FALSE",
                 I_Spare11 := "FALSE",
                 I_Spare12 := "FALSE",
                 I_Spare13 := "FALSE",
                 I_Spare14 := "FALSE",
                 H_IAnim => #H_HMI.H_IAnim);
END_REGION

REGION Network 60: *** 5.1 - Interlocks **** Reset interlock OP if inactive timeout or logout
   // Reset interlock OP if inactive timeout or logout
   INTL:
   #ResetOP := #AutoSel AND #OP_Selected;
   IF #ResetOP THEN
       #OP_Selected := FALSE;
       #OP_TimeoutInput := FALSE;
       #Request_Logout := FALSE;
       #GroupInterlock := 0;
       #OP_ScreenWanted := 1;
   END_IF;
END_REGION

REGION Network 61: *** 4.4 Machine Status, calculated *** Attempt to activate the OP, pressing F1-F4
   // Attempt to activate the OP, pressing F1-F4, changing to a screen
   // F2 is the logout function
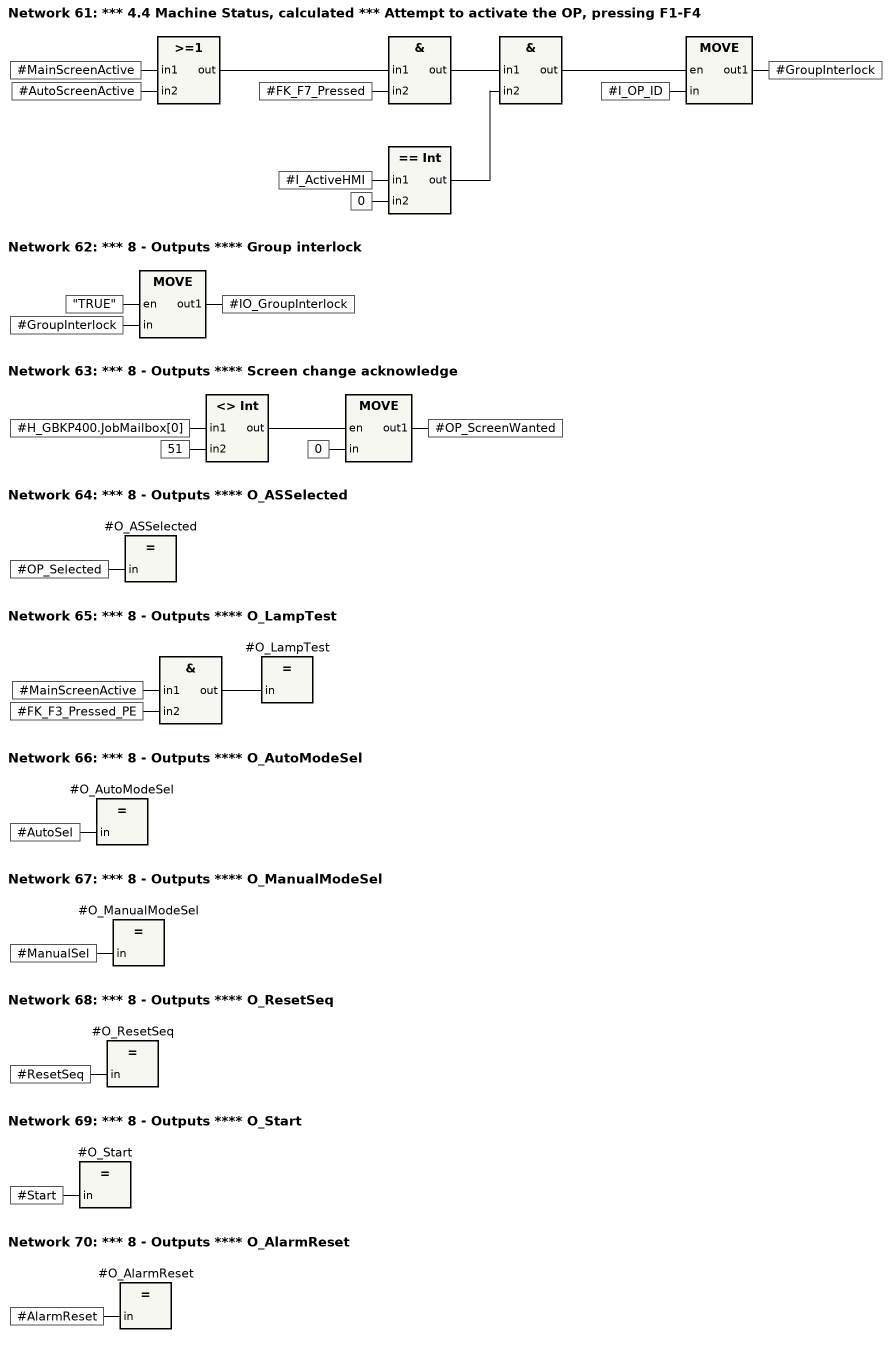
   IF (#MainScreenActive OR #AutoScreenActive) AND #FK_F7_Pressed AND (#I_ActiveHMI = 0) THEN
       #GroupInterlock := #I_OP_ID;
   END_IF;
END_REGION

REGION Network 62: *** 8 - Outputs **** Group interlock
   // Group interlock
   IF "TRUE" THEN #IO_GroupInterlock := #GroupInterlock; END_IF;
END_REGION

REGION Network 63: *** 8 - Outputs **** Screen change acknowledge
   // Screen change acknowledge
   IF #H_GBKP400.JobMailbox[0] <> 51 THEN #OP_ScreenWanted := 0; END_IF;
END_REGION

REGION Network 64: *** 8 - Outputs **** O_ASSelected
   // O_ASSelected
   #O_ASSelected := #OP_Selected;
END_REGION

REGION Network 65: *** 8 - Outputs **** O_LampTest
   // O_LampTest
   #O_LampTest := #MainScreenActive AND #FK_F3_Pressed_PE;
END_REGION

REGION Network 66: *** 8 - Outputs **** O_AutoModeSel
   // O_AutoModeSel
   #O_AutoModeSel := #AutoSel;
END_REGION

REGION Network 67: *** 8 - Outputs **** O_ManualModeSel
   // O_ManualModeSel
   #O_ManualModeSel := #ManualSel;
END_REGION

REGION Network 68: *** 8 - Outputs **** O_ResetSeq
   // O_ResetSeq
   // O_ResetTM identical to O_ResetSeq
   #O_ResetSeq := #ResetSeq;
END_REGION

REGION Network 69: *** 8 - Outputs **** O_Start
   // O_Start
   #O_Start := #Start;
END_REGION

REGION Network 70: *** 8 - Outputs **** O_AlarmReset
   // O_AlarmReset
   #O_AlarmReset := #AlarmReset;
END_REGION

REGION Network 71: *** 8 - Outputs **** O_HighSpeed
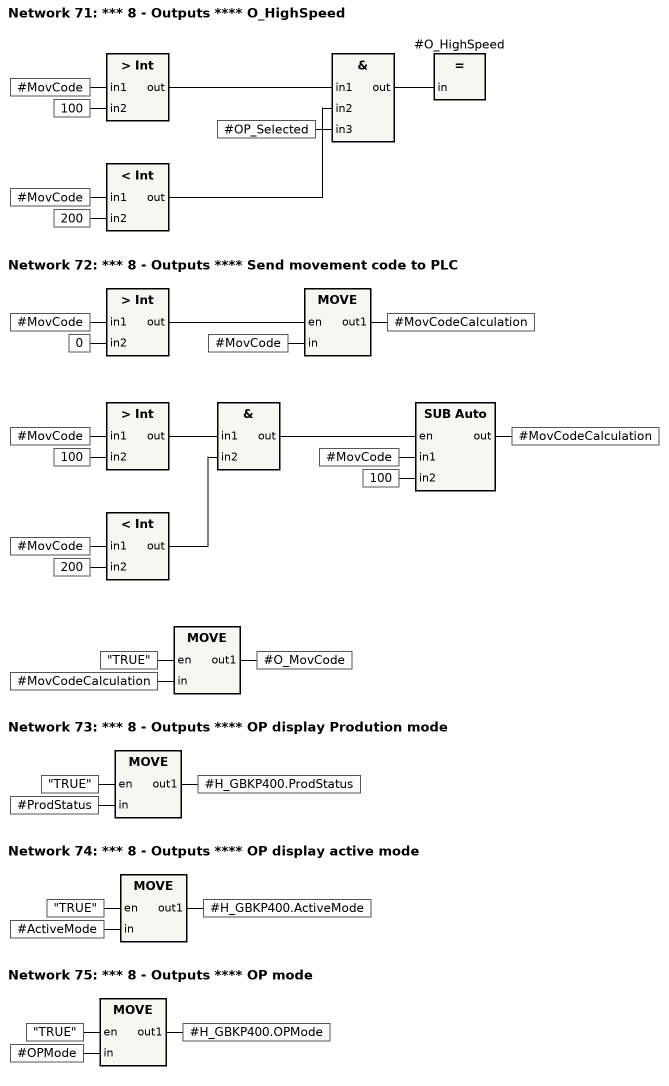
   #O_HighSpeed := (#MovCode > 100) AND (#MovCode < 200) AND #OP_Selected;
END_REGION

REGION Network 72: *** 8 - Outputs **** Send movement code to PLC
   // Send movement code to PLC
   IF #MovCode > 0 THEN #MovCodeCalculation := #MovCode; END_IF;
   IF (#MovCode > 100) AND (#MovCode < 200) THEN #MovCodeCalculation := #MovCode - 100; END_IF;
   IF "TRUE" THEN #O_MovCode := #MovCodeCalculation; END_IF;
END_REGION

REGION Network 73: *** 8 - Outputs **** OP display Prodution mode
   // OP display Prodution mode
   IF "TRUE" THEN #H_GBKP400.ProdStatus := #ProdStatus; END_IF;
END_REGION

REGION Network 74: *** 8 - Outputs **** OP display active mode
   // OP display active mode
   IF "TRUE" THEN #H_GBKP400.ActiveMode := #ActiveMode; END_IF;
END_REGION

REGION Network 75: *** 8 - Outputs **** OP mode
   // OP mode
   IF "TRUE" THEN #H_GBKP400.OPMode := #OPMode; END_IF;
END_REGION
END_FUNCTION_BLOCK
